// TwinCAT 3 PLC project PLC
// ProgramVersion: 3.1.4026.20
// CompilerDefines: VISU_USEPROPERTYINFO
// libraries:
//   SPT Base Types, * (Beckhoff Automation LLC)
//   SPT Components, * (Beckhoff Automation LLC)
//   SPT Diagnostic, * (Beckhoff Automation LLC)
//   SPT EtherCat, * (Beckhoff Automation LLC)
//   SPT Event Logger, * (Beckhoff Automation LLC)
//   SPT Motion Control, * (Beckhoff Automation LLC)
//   SPT Utilities, * (Beckhoff Automation LLC)
//   Tc2_MC2, * (Beckhoff Automation GmbH)
//   Tc2_MC2_Camming, * (Beckhoff Automation GmbH)
//   Tc2_Standard, * (Beckhoff Automation GmbH)
//   Tc2_System, * (Beckhoff Automation GmbH)
//   Tc2_Utilities, * (Beckhoff Automation GmbH)
//   Tc3_EventLogger, * (Beckhoff Automation GmbH)
//   Tc3_MC2_AdvancedHoming, * (Beckhoff Automation GmbH)
//   Tc3_McCollisionAvoidance, * (Beckhoff Automation GmbH)
//   Tc3_McCoordinatedMotion, * (Beckhoff Automation GmbH)
//   Tc3_PackML_V3, * (Beckhoff Automation GmbH)
// project tree:
//   / GlobalTextList.TcGTLO (not stored), PlcTask.TcTTO (not stored), VisualizationManager.TcVMO (not stored)
//   GVLs/ GVL.TcGVL (not stored)
//   POUs/BeltIndexer/ FB_DataSetFifo.TcPOU (not stored), FB_BeltIndexer.TcPOU
//   POUs/ Machine.TcPOU, MAIN.TcPOU (not stored)
//   VISUs/ Visualization.TcVIS (not stored)
// real-time tasks:
//   TASK PlcTask: cycle T#1ms, priority 20, ADS port 350
//   TASK Job Task: cycle default, priority 32
// motion (NC):
//   TASK NC-Task 1 SAF: cycle T#2ms, priority 4, ADS port 501
//   TASK NC-Task 1 SVB: cycle T#10ms, priority 8, ADS port 511
//   AXIS Cam_Master (id 3)
//     General: UnitName=°, UnitFlags=#x00000004
//     Dynamic: Acceleration=15000, Deceleration=15000, Jerk=73844.676
//     Velo: RefSearch=164.09928, RefSync=164.09928, SlowManual=820.4964, FastManual=4922.9784, Fast=16409.928, Maximum=16409.928
//     OtherSettings: AllowMotionCmdToSlave=true
//     encoder EncType=19
//       EncPara: ScaleFactorNumerator=360, ScaleFactorDenominator=1048576, MaxCount=#xffffffff
//     drive DrvType=16
//       DrvPara: MaxCount=#xffffffff, DriveControlDWord=#x00020100
//         Analog: VeloReferenz=18050.9208, VeloScale=71.5255737304688, TorqueSetpointScale=10, ScaleFactorActTorque=0.1
//         TimeComp: TaskDelayCycles=1
//     controller CtrType=1
//       CtrPara: PriorControlFactor=1
//         Observer: BandWidth=20
//   AXIS TouchProbe (id 4)
//     General: UnitName=°
//     Dynamic: Acceleration=15000, Deceleration=15000, Jerk=73844.676
//     Velo: RefSearch=164.09928, RefSync=164.09928, SlowManual=820.4964, FastManual=4922.9784, Fast=16409.928, Maximum=16409.928
//     OtherSettings: AllowMotionCmdToSlave=true
//     encoder EncType=19
//       EncPara: ScaleFactorNumerator=360, ScaleFactorDenominator=1048576, Inverse=true, MaxCount=#xffffffff
//     drive DrvType=16
//       DrvPara: Inverse=true, MaxCount=#xffffffff, DriveControlDWord=#x00020100
//         Analog: VeloReferenz=18050.9208, VeloScale=71.5255737304688, TorqueSetpointScale=10, ScaleFactorActTorque=0.1
//         TimeComp: TaskDelayCycles=1
//     controller CtrType=1
//       CtrPara: PriorControlFactor=1
//         Observer: BandWidth=20
//   AXIS Cam_Slave (id 5)
//     General: UnitName=°, UnitFlags=#x00000004
//     Dynamic: Acceleration=15000, Deceleration=15000, Jerk=71760.627
//     Velo: RefSearch=159.46806, RefSync=159.46806, SlowManual=797.3403, FastManual=4784.0418, Fast=15946.806, Maximum=15946.806
//     OtherSettings: AllowMotionCmdToSlave=true
//     encoder EncType=19
//       EncPara: ScaleFactorNumerator=360, ScaleFactorDenominator=1048576, Inverse=true, MaxCount=#xffffffff
//     drive DrvType=16
//       DrvPara: Inverse=true, MaxCount=#xffffffff, DriveControlDWord=#x00020100
//         Analog: VeloReferenz=17541.4866, VeloScale=71.5255737304688, TorqueSetpointScale=10, ScaleFactorActTorque=0.1
//         TimeComp: TaskDelayCycles=1
//     controller CtrType=1
//       CtrPara: PriorControlFactor=1
//         PosDiffControl: Enable=false, Range=10
//         Observer: BandWidth=20
// I/O:
//   DEVICE Device 2 (EtherCAT), AmsNetId 5.151.68.96.3.1
//     Term 1 (EK1200) [EK1200-5000 EtherCAT Power supply (2A E-Bus)]
//       Term 2 (EL2911) [EL2911, Potential supply terminal (10 A) with 4 Ch. Safety Inputs, TwinSAFE]
//         modules: Module 2 (FSOUT), Module 3 (DEVICEIO), Module 4 (FSLOGIC)
//       Term 3 (EL1859) [EL1859 8Ch. Dig. Input 24V, 3ms, 8Ch. Dig. Output 24V, 0.5A]
//       Term 4 (EL9011) [EL9011 End Terminal]
//   DEVICE Device 3 (EtherCAT), AmsNetId 5.151.68.96.4.1
//     Term 5 (AX8620-0000-0103) [AX8620-0000-0103]
//       Drive 6 (AX8206-0200-0106) [AX8206-0200-0106 (2Ch. 6A servo axis, safe-motion)]
//         modules: Device, Device, Device, Device, Device, Device, Device, Device, Device, Device, Device (Safety), Device, Device, Device, Device, Device, Device, Device, Device, Device, Device, Device, Device, Device, Device, Device, Device, Device, Device, Device, Device, Ch A, Ch A, Ch A, Ch A, Ch A, Ch A, Ch A, Ch A, Ch A, Ch A, Ch A, Ch A, Ch A, Ch A, Ch A, Ch A, Ch A, Ch A, Ch A, Ch A, Ch A, Ch A, Ch A, Ch A, Ch A, Ch A, Ch A, Ch B, Ch B, Ch B, Ch B, Ch B, Ch B, Ch B, Ch B, Ch B, Ch B, Ch B, Ch B, Ch B, Ch B, Ch B, Ch B, Ch B, Ch B, Ch B, Ch B, Ch B, Ch B, Ch B, Ch B, Ch B, Ch B, Ch B
//         startup 12992:1 := 414D383032322D78447831 // Ch A Motor parameters / Configured motor type
//         startup 24768:0 := FEFF // Ch A Interpolation sub mode select
//         startup 13000:5 := 0200 // Ch A Motor thermal model / Reaction
//         startup 13000:6 := 0000C841 // Ch A Motor thermal model / Partial fraction factor
//         startup 12992:12 := 0000FA45 // Ch A Motor parameters / Motor rated speed
//         startup 12992:13 := E561313F // Ch A Motor parameters / Motor rated torque
//         startup 24694:0 := 20030000 // Ch A Motor standstill torque
//         startup 24800:0 := D007 // Ch A Positive torque/force limit value
//         startup 24801:0 := D007 // Ch A Negative torque/force limit value
//         startup 12288:6 := 4158383230362D303230302D30303030 // Ch A AxisMain parameters / Configured drive type
//         startup 12867:1 := 0000C03F // Ch A TorqueCtrl parameters / Configured channel rated current
//         startup 12867:2 := 00009040 // Ch A TorqueCtrl parameters / Configured channel peak current
//         startup 12867:7 := 77BE1F40 // Ch A TorqueCtrl parameters / Iuvw max sum
//         startup 24672:0 := 08 // Ch A Modes of operation
//         startup 13023:0 := 0000 // Ch A Motor control mode
//         startup 12998:1 := 2D6F0C3D // Ch A Motor commutation monitoring parameters / Speed threshold
//         startup 12864:1 := 88E9D742 // Ch A TorqueCtrl parameters mappable / Torque control proportional gain q
//         startup 12864:2 := 8A0E7C39 // Ch A TorqueCtrl parameters mappable / Torque control integral action time q
//         startup 12608:1 := 7298793C // Ch A VeloCtrl parameters mappable / Velocity control proportional gain
//         startup 12608:2 := 6F12033C // Ch A VeloCtrl parameters mappable / Velocity control integral action time
//         startup 12608:3 := 00980546 // Ch A VeloCtrl parameters mappable / Bipolar velocity limit value
//         startup 12992:15 := 0100 // Ch A Motor parameters / Motor temperature sensor connection
//         startup 12611:4 := 0400 // Ch A VeloCtrl observer / Observer type
//         startup 24672:0 := 08 // Ch A Modes of operation
//         startup 12296:2 := 00 // Ch A AxisMain parameters encoder direction / Primary encoder direction
//         startup 14016:1 := 414D383032322D78447831 // Ch B Motor parameters / Configured motor type
//         startup 26816:0 := FEFF // Ch B Interpolation sub mode select
//         startup 14024:5 := 0200 // Ch B Motor thermal model / Reaction
//         startup 14024:6 := 0000C841 // Ch B Motor thermal model / Partial fraction factor
//         startup 14016:12 := 0000FA45 // Ch B Motor parameters / Motor rated speed
//         startup 14016:13 := E561313F // Ch B Motor parameters / Motor rated torque
//         startup 26742:0 := 20030000 // Ch B Motor standstill torque
//         startup 26848:0 := D007 // Ch B Positive torque/force limit value
//         startup 26849:0 := D007 // Ch B Negative torque/force limit value
//         startup 13312:6 := 4158383230362D303230302D30303030 // Ch B AxisMain parameters / Configured drive type
//         startup 13891:1 := 0000C03F // Ch B TorqueCtrl parameters / Configured channel rated current
//         startup 13891:2 := 00009040 // Ch B TorqueCtrl parameters / Configured channel peak current
//         startup 13891:7 := 77BE1F40 // Ch B TorqueCtrl parameters / Iuvw max sum
//         startup 26720:0 := 08 // Ch B Modes of operation
//         startup 14047:0 := 0000 // Ch B Motor control mode
//         startup 14022:1 := 2D6F0C3D // Ch B Motor commutation monitoring parameters / Speed threshold
//         startup 13888:1 := 88E9D742 // Ch B TorqueCtrl parameters mappable / Torque control proportional gain q
//         startup 13888:2 := 8A0E7C39 // Ch B TorqueCtrl parameters mappable / Torque control integral action time q
//         startup 13632:1 := 7298793C // Ch B VeloCtrl parameters mappable / Velocity control proportional gain
//         startup 13632:2 := 6F12033C // Ch B VeloCtrl parameters mappable / Velocity control integral action time
//         startup 13632:3 := 00980546 // Ch B VeloCtrl parameters mappable / Bipolar velocity limit value
//         startup 14016:15 := 0100 // Ch B Motor parameters / Motor temperature sensor connection
//         startup 13635:4 := 0400 // Ch B VeloCtrl observer / Observer type
//         startup 26720:0 := 08 // Ch B Modes of operation
//         startup 13320:2 := 00 // Ch B AxisMain parameters encoder direction / Primary encoder direction
//       Term 7 (AX8831-0000-0201) [AX8831-0000-0201]
//         Drive 8 (AMP8000-0030-0106) [AMP8000-0030-0106 (distributed servo drive, STO, safe motion)]
//           modules: Device, Device, Device, Device, Device, Device, Device, Device, Device, Device, Device (Safety), Device, Device, Device, Device, Device, Device, Device, Device, Device, Device, Device, Device, Device, Device, Device, Device, Device, Device, Device, Device, Ch A, Ch A, Ch A, Ch A, Ch A, Ch A, Ch A, Ch A, Ch A, Ch A, Ch A, Ch A, Ch A, Ch A, Ch A, Ch A, Ch A, Ch A, Ch A, Ch A, Ch A, Ch A, Ch A, Ch A, Ch A, Ch A, Ch A
//           startup 12992:1 := 414D50383034322D4A787831 // Ch A Motor parameters / Configured motor type
//           startup 24768:0 := FEFF // Ch A Interpolation sub mode select
//           startup 13000:5 := 0200 // Ch A Motor thermal model / Reaction
//           startup 13000:6 := 0000C841 // Ch A Motor thermal model / Partial fraction factor
//           startup 12992:12 := 00C0DA45 // Ch A Motor parameters / Motor rated speed
//           startup 12992:13 := 8941803F // Ch A Motor parameters / Motor rated torque
//           startup 24694:0 := 000F0000 // Ch A Motor standstill torque
//           startup 24800:0 := D007 // Ch A Positive torque/force limit value
//           startup 24801:0 := D007 // Ch A Negative torque/force limit value
//           startup 12288:6 := 414D50383030302D303033302D30303030 // Ch A AxisMain parameters / Configured drive type
//           startup 12867:1 := CDCCCC40 // Ch A TorqueCtrl parameters / Configured channel rated current
//           startup 12867:2 := 00009041 // Ch A TorqueCtrl parameters / Configured channel peak current
//           startup 12867:7 := F4FD5440 // Ch A TorqueCtrl parameters / Iuvw max sum
//           startup 24672:0 := 08 // Ch A Modes of operation
//           startup 13023:0 := 0000 // Ch A Motor control mode
//           startup 12998:1 := 0834053D // Ch A Motor commutation monitoring parameters / Speed threshold
//           startup 12864:1 := 84C3B441 // Ch A TorqueCtrl parameters mappable / Torque control proportional gain q
//           startup 12864:2 := 8A0E7C39 // Ch A TorqueCtrl parameters mappable / Torque control integral action time q
//           startup 12608:1 := B379FC3D // Ch A VeloCtrl parameters mappable / Velocity control proportional gain
//           startup 12608:2 := 6F12033C // Ch A VeloCtrl parameters mappable / Velocity control integral action time
//           startup 12608:3 := 00980546 // Ch A VeloCtrl parameters mappable / Bipolar velocity limit value
//           startup 12992:15 := 0100 // Ch A Motor parameters / Motor temperature sensor connection
//           startup 12611:4 := 0400 // Ch A VeloCtrl observer / Observer type
//           startup 24672:0 := 08 // Ch A Modes of operation
//           startup 12296:2 := 00 // Ch A AxisMain parameters encoder direction / Primary encoder direction
// variable links:
//   Device 2 (EtherCAT) <-> Device 3 (EtherCAT)/Term 5 (AX8620-0000-0103)/Drive 6 (AX8206-0200-0106)
//     Term 1 (EK1200)/Term 2 (EL2911)/ConnectionInputs/Message_20 TxPDO <-> Device (Safety)/FSoE Slave Connection 1 Master Message/FSOE
//     Term 1 (EK1200)/Term 2 (EL2911)/ConnectionOutputs/Message_20 RxPDO <-> Device (Safety)/FSoE Slave Connection 1 Slave Message/FSOE
//   Device 2 (EtherCAT) <-> Device 3 (EtherCAT)/Term 5 (AX8620-0000-0103)/Term 7 (AX8831-0000-0201)/Drive 8 (AMP8000-0030-0106)
//     Term 1 (EK1200)/Term 2 (EL2911)/ConnectionInputs/Message_21 TxPDO <-> Device (Safety)/FSoE Connection 1 Receive Message/Message_1
//     Term 1 (EK1200)/Term 2 (EL2911)/ConnectionOutputs/Message_21 RxPDO <-> Device (Safety)/FSoE Connection 1 Send Message/Message_1
//   Device 3 (EtherCAT) <-> Device 3 (EtherCAT)/Term 5 (AX8620-0000-0103)
//     Term 5 (AX8620-0000-0103)/Drive 6 (AX8206-0200-0106)/Device/DeviceMain Outputs/Power supply controlword <-> PSM Controlword for axis/Controlword for axis
//     Term 5 (AX8620-0000-0103)/Term 7 (AX8831-0000-0201)/PSM Controlword out/Controlword out <-> PSM Controlword for axis/Controlword for axis
//   Device 3 (EtherCAT) <-> Device 3 (EtherCAT)/Term 5 (AX8620-0000-0103)/Term 7 (AX8831-0000-0201)
//     Term 5 (AX8620-0000-0103)/Term 7 (AX8831-0000-0201)/Drive 8 (AMP8000-0030-0106)/Device/DeviceMain Outputs/Power supply controlword <-> PSM Controlword in/Controlword 1 in
//   NC-Task 1 SAF/Axes/Cam_Master <-> Device 3 (EtherCAT)/Term 5 (AX8620-0000-0103)/Drive 6 (AX8206-0200-0106)
//     Drive/Inputs/In/nDataIn1 <-> Ch A/Ch A PositionControl Inputs/Ch A Following error actual value
//     Drive/Inputs/In/nDataIn3[0] <-> Ch A/Ch A TorqueControl Inputs/Ch A Torque/force actual value
//     Drive/Inputs/In/nDcOutputTime <-> InfoData/DcOutputShift
//     Drive/Inputs/In/nState1 <-> Ch A/Ch A AxisMain Inputs/Ch A Statusword
//     Drive/Inputs/In/nState2 <-> Ch A/Ch A AxisMain Inputs/Ch A Statusword @bit 8
//     Drive/Inputs/In/nState4 @bit 1 <-> WcState/InputToggle0
//     Drive/Inputs/In/nState4 <-> WcState/WcState0
//     Drive/Outputs/Out/nCtrl1 <-> Ch A/Ch A AxisMain Outputs/Ch A Controlword
//     Drive/Outputs/Out/nCtrl2 <-> Ch A/Ch A AxisMain Outputs/Ch A Controlword @bit 8
//     Drive/Outputs/Out/nDataOut1 <-> Ch A/Ch A Interpolator Outputs/Ch A Target position
//     Drive/Outputs/Out/nDataOut2 <-> Ch A/Ch A Interpolator Outputs/Ch A Target velocity
//     Enc/Inputs/In/nDataIn1 <-> Ch A/Ch A AxisMain Inputs/Ch A Position actual value
//     Enc/Inputs/In/nDcInputTime <-> InfoData/DcInputShift
//     Enc/Inputs/In/nState2 @bit 5 <-> Ch A/Ch A AxisMain Inputs/Position actual value invalid
//     Enc/Inputs/In/nState4 @bit 1 <-> WcState/InputToggle0
//     Enc/Inputs/In/nState4 <-> WcState/WcState0
//   NC-Task 1 SAF/Axes/Cam_Slave <-> Device 3 (EtherCAT)/Term 5 (AX8620-0000-0103)/Term 7 (AX8831-0000-0201)/Drive 8 (AMP8000-0030-0106)
//     Drive/Inputs/In/nDataIn1 <-> Ch A/Ch A PositionControl Inputs/Ch A Following error actual value
//     Drive/Inputs/In/nDataIn3[0] <-> Ch A/Ch A TorqueControl Inputs/Ch A Torque/force actual value
//     Drive/Inputs/In/nDcOutputTime <-> InfoData/DcOutputShift
//     Drive/Inputs/In/nState1 <-> Ch A/Ch A AxisMainAMP Inputs/Ch A Statusword
//     Drive/Inputs/In/nState2 <-> Ch A/Ch A AxisMainAMP Inputs/Ch A Statusword @bit 8
//     Drive/Inputs/In/nState4 @bit 1 <-> WcState/InputToggle0
//     Drive/Inputs/In/nState4 <-> WcState/WcState0
//     Drive/Outputs/Out/nCtrl1 <-> Ch A/Ch A AxisMainAMP Outputs/Ch A Controlword
//     Drive/Outputs/Out/nCtrl2 <-> Ch A/Ch A AxisMainAMP Outputs/Ch A Controlword @bit 8
//     Drive/Outputs/Out/nDataOut1 <-> Ch A/Ch A Interpolator Outputs/Ch A Target position
//     Drive/Outputs/Out/nDataOut2 <-> Ch A/Ch A Interpolator Outputs/Ch A Target velocity
//     Enc/Inputs/In/nDataIn1 <-> Ch A/Ch A AxisMainAMP Inputs/Ch A Position actual value
//     Enc/Inputs/In/nDcInputTime <-> InfoData/DcInputShift
//     Enc/Inputs/In/nState2 @bit 5 <-> Ch A/Ch A AxisMainAMP Inputs/Position actual value invalid
//     Enc/Inputs/In/nState4 @bit 1 <-> WcState/InputToggle0
//     Enc/Inputs/In/nState4 <-> WcState/WcState0
//   NC-Task 1 SAF/Axes/TouchProbe <-> Device 3 (EtherCAT)/Term 5 (AX8620-0000-0103)/Drive 6 (AX8206-0200-0106)
//     Drive/Inputs/In/nDataIn1 <-> Ch B/Ch B PositionControl Inputs/Ch B Following error actual value
//     Drive/Inputs/In/nDataIn3[0] <-> Ch B/Ch B TorqueControl Inputs/Ch B Torque/force actual value
//     Drive/Inputs/In/nDcOutputTime <-> InfoData/DcOutputShift
//     Drive/Inputs/In/nState1 <-> Ch B/Ch B AxisMain Inputs/Ch B Statusword
//     Drive/Inputs/In/nState2 <-> Ch B/Ch B AxisMain Inputs/Ch B Statusword @bit 8
//     Drive/Inputs/In/nState4 @bit 1 <-> WcState/InputToggle0
//     Drive/Inputs/In/nState4 <-> WcState/WcState0
//     Drive/Outputs/Out/nCtrl1 <-> Ch B/Ch B AxisMain Outputs/Ch B Controlword
//     Drive/Outputs/Out/nCtrl2 <-> Ch B/Ch B AxisMain Outputs/Ch B Controlword @bit 8
//     Drive/Outputs/Out/nDataOut1 <-> Ch B/Ch B Interpolator Outputs/Ch B Target position
//     Drive/Outputs/Out/nDataOut2 <-> Ch B/Ch B Interpolator Outputs/Ch B Target velocity
//     Enc/Inputs/In/nDataIn1 <-> Ch B/Ch B AxisMain Inputs/Ch B Position actual value
//     Enc/Inputs/In/nDcInputTime <-> InfoData/DcInputShift
//     Enc/Inputs/In/nState2 @bit 5 <-> Ch B/Ch B AxisMain Inputs/Position actual value invalid
//     Enc/Inputs/In/nState4 @bit 1 <-> WcState/InputToggle0
//     Enc/Inputs/In/nState4 <-> WcState/WcState0
//   PLC/PLC Instance <-> Device 2 (EtherCAT)/Term 1 (EK1200)/Term 2 (EL2911)
//     PlcTask Inputs/MAIN.SafetyEstop.InfoData/Diag <-> TwinSAFE Group Info Data/TwinSafeGroup1 Info Data/Diag
//     PlcTask Inputs/MAIN.SafetyEstop.InfoData/State <-> TwinSAFE Group Info Data/TwinSafeGroup1 Info Data/State
//     PlcTask Inputs/MAIN.SafetyGroup_Main.InfoData/Diag <-> TwinSAFE Group Info Data/TwinSafeGroup1 Info Data/Diag
//     PlcTask Inputs/MAIN.SafetyGroup_Main.InfoData/State <-> TwinSAFE Group Info Data/TwinSafeGroup1 Info Data/State
//     PlcTask Outputs/MAIN.SafetyFBReset <-> StandardOutputs/Standard In Var 8
//     PlcTask Outputs/MAIN.SafetyGroupAutoReset.Reset <-> StandardOutputs/Standard In Var 1
//     PlcTask Outputs/MAIN.SafetyGroup_Main.Run <-> StandardOutputs/Standard In Var 2
//   PLC/PLC Instance <-> Device 3 (EtherCAT)/Term 5 (AX8620-0000-0103)/Term 7 (AX8831-0000-0201)/Drive 8 (AMP8000-0030-0106)
//     PlcTask Outputs/MAIN.SafetyGroupAutoReset.Reset <-> Device (Safety)/Standard Outputdata/Standard In Var 3
//     PlcTask Outputs/MAIN.SafetyGroup_Main.Run <-> Device (Safety)/Standard Outputdata/Standard In Var 2
//   PLC/PLC Instance <-> NC-Task 1 SAF/Axes/TouchProbe
//     PlcTask Inputs/MAIN.Machine.BeltIndexer.BeltAxis.BasicAxis._Axis.NcToPlc <-> Outputs/ToPlc
//     PlcTask Outputs/MAIN.Machine.BeltIndexer.BeltAxis.BasicAxis._Axis.PlcToNc <-> Inputs/FromPlc

// ---- POUs/Machine.TcPOU
FUNCTION_BLOCK Machine EXTENDS FB_PackML_BaseModule
VAR
	BeltIndexer		: FB_BeltIndexer;
END_VAR

METHOD PROTECTED HMIPermissions
AllowHMIControl(TRUE);
END_METHOD

(* Basic module initialization logic*)
METHOD PROTECTED Initialize : BOOL
Initialize := FALSE;
CASE DescendantSequenceState OF
	0:
		//RegisterSubmodule(SubModule	:= CamModule);
		RegisterSubmodule(SubModule	:= BeltIndexer);
		DescendantSequenceState := DescendantSequenceState + 10;

	10:
		IF SUPER^.Initialize() THEN
			Initialize := TRUE;
		END_IF
END_CASE
END_METHOD

END_FUNCTION_BLOCK

// ---- POUs/BeltIndexer/FB_BeltIndexer.TcPOU
FUNCTION_BLOCK FB_BeltIndexer EXTENDS FB_PackML_BaseModule
VAR
	BeltAxis	: FB_Component_BasicAxis;

	fbFifo 				: FB_DataSetFifo := ( bOverwrite := TRUE );
	arrBuffer 			: ARRAY[0..MAX_BUFFER_SIZE] OF BYTE; (* Buffer memory used by FB_MemRingBuffer function block *)

	NewRecordedPosition	: LREAL;
	OldRecordedPosition	: LREAL;

	TON_Dwell	: TON;
END_VAR

//! @summary This method contains code which will execute when this PackML module is in the <b>Aborting</b> state
METHOD PROTECTED Aborting
VAR
	i				: UDINT;
	SubModulesReady : BOOL := TRUE;
END_VAR
CASE DescendantSequenceState OF
	0:
		NoStateTasksToComplete := FALSE;
		DescendantSequenceState := DescendantSequenceState + 10;

	10:
		IF BeltAxis.Disable() THEN
			NewRecordedPosition		:= 0;
			OldRecordedPosition		:= 0;
			StateTasksComplete 		:= TRUE;
			DescendantSequenceState := DescendantSequenceState + 10;
		END_IF

	//20:	

	20:
		StateTasksComplete := TRUE;
END_CASE

SUPER^.Aborting();
END_METHOD

//! @summary This method contains code which will execute when this PackML module is in the <b>Clearing</b> state
METHOD PROTECTED Clearing
VAR
	i				: UDINT;
	SubModulesReady : BOOL := TRUE;
END_VAR

VAR_INST

END_VAR

(*! <description> <b>Note:</b> The <i>Clear</i> command can also be thought of as a <i>fault reset</i> depite the ambiguity in the naming of the <i>Reset</i> state. 
<table> 
	<tr>
		<th> Previous State </th>
		<th> Transition In </th>
		<th> Transition Out </th>
		<th> Next State  </th> 
	</tr>
	<tr>
		<td> Aborted </td>
		<td> Clear Command </td> 
		<td> State Complete </td>
		<td> Stopped </td> 
	</tr>
</table>
This method is called as required by <c>StateControl()</c>
</description> 

*)
// CASE _CurrentMode OF
// 	E_PMLUnitMode.ePMLUnitMode_Production:
		CASE DescendantSequenceState OF
			0: //Init
				NoStateTasksToComplete := FALSE;

				//Reset Axes and  CA Group
				BeltAxis.Reset();
				DescendantSequenceState := DescendantSequenceState + 10;

			10: // Done	
				StateTasksComplete := TRUE;
		END_CASE

// END_CASE

SUPER^.Clearing();
END_METHOD

METHOD CyclicLogic
VAR_INPUT
END_VAR
SUPER^.CyclicLogic();

fbFifo();
TON_Dwell();
END_METHOD

//! @summary This method contains code which will execute when this PackML module is in the <b>Execute</b> state
METHOD PROTECTED Execute
VAR
	i : UDINT;
END_VAR
(*CASE _CurrentMode OF
	E_PMLUnitMode.ePMLUnitMode_Production:


	E_PMLUnitMode.ePMLUnitMode_Manual:
		; //Insert logic for Manual Mode here
END_CASE	*)

CASE DescendantSequenceState OF
	0:	// Start Moving
		BeltAxis.MoveVelocity(250, TRUE);
		DescendantSequenceState	:= DescendantSequenceState + 10;

	10: // Start buffering positions and moving to them
		IF fbFifo.nCount > 0 THEN
			fbFifo.A_Get(out => OldRecordedPosition);
			BeltAxis.MoveAbsolute(OldRecordedPosition + 440.0, TRUE);
			DescendantSequenceState	:= DescendantSequenceState + 10;
		END_IF
		
	20: // Look for trigger
		IF ton_dwell.Q THEN
			TON_Dwell.IN			:= FALSE;
			fbFifo.A_Remove();
			IF fbFifo.nCount > 0 THEN
				DescendantSequenceState	:= 10;
			ELSE
				DescendantSequenceState	:= 0;
			END_IF
		ELSIF BeltAxis.InPosition AND (ABS(BeltAxis.SetPosition - (OldRecordedPosition + 440)) < 1) THEN
			Ton_Dwell.IN	:= TRUE;
		END_IF

END_CASE

//run this with new recorded positions from touchprobe	
//fbFifo.A_Add(In := NewRecordedPosition);
END_METHOD

(* Basic module initialization logic*)
METHOD PROTECTED Initialize : BOOL
Initialize := FALSE;
CASE DescendantSequenceState OF
	0:
		RegisterComponent(Component := BeltAxis);
		DescendantSequenceState := DescendantSequenceState + 10;

	10: // Touch Probe Configuration
		TON_Dwell.PT					:= T#500MS;
		DescendantSequenceState 		:= DescendantSequenceState + 10;

	20:
		IF SUPER^.Initialize() THEN
			DescendantSequenceState := DescendantSequenceState + 10;
		END_IF

	30:
		Initialize := TRUE;
END_CASE
END_METHOD

METHOD PROTECTED Resetting
VAR_INST
	i			 : UDINT;
END_VAR
// CASE _CurrentMode OF
// 	E_PMLUnitMode.ePMLUnitMode_Production:
		CASE DescendantSequenceState OF
			0: //Init
				i					   := 1;
				NoStateTasksToComplete := FALSE;
				DescendantSequenceState := DescendantSequenceState + 10;

			10: //Enable Axes
				IF BeltAxis.Enable() THEN
					DescendantSequenceState := DescendantSequenceState + 10;
				END_IF

			20:	// Home Axis
				IF BeltAxis.Home() THEN
					DescendantSequenceState := DescendantSequenceState + 10;
				END_IF
	
			30: // Clear Buffer
				fbFifo.A_Reset();
				DescendantSequenceState := DescendantSequenceState + 10;

			40: //Clearing complete
				StateTasksComplete := TRUE;

		END_CASE
// END_CASE

SUPER^.Resetting();
END_METHOD

METHOD PROTECTED Starting
VAR_INST
	i		  : UDINT;
END_VAR
//CASE _CurrentMode OF
//	E_PMLUnitMode.ePMLUnitMode_Production:
		CASE DescendantSequenceState OF
			0:
				NoStateTasksToComplete	:= FALSE;
				DescendantSequenceState := 10;
				i						:= 1;

			10: //Set Axis Parameters
				BeltAxis.Velocity		:= 250;
				BeltAxis.Acceleration	:= 1000;
				BeltAxis.Deceleration	:= 1000;
				BeltAxis.Jerk			:= 1000;
				DescendantSequenceState := DescendantSequenceState + 10;

			20: // Start Touchprobe and clear buffer
				DescendantSequenceState 	:= DescendantSequenceState + 10;
				
			30: // Finsihed
				StateTasksComplete 		:= TRUE;

		END_CASE

	//E_PMLUnitMode.ePMLUnitMode_Manual:
//END_CASE

SUPER^.Starting();
END_METHOD

END_FUNCTION_BLOCK
